TYPE CM_Valve_SIM :
STRUCT
END_STRUCT
END_TYPE

(* stored: Version 1.1.0.1, ProductVersion 3.1.4024.12
   DUT CM_Valve_SIM: Id {dbeabb42-d200-4016-aa1e-ad2d5b0e180c} *)
